# B&R Automation Studio project ACP180_Test
Automation Studio 4.12.5.95 SP; technology packages: mappMotion 5.26.1, mappView 5.24.1

## Configuration APC910

CPU 5PC900.TS17-00, AutomationRuntime M4.93, Build 4.1.2, Safety 0.0, Vc V4.72.6

### Task classes (Cpu.sw)
```
Cyclic#1 (cycle 800 us, tolerance 0 us):
  ShCamCtr <- Prog.ShCamCtr.prg
  StartMove <- Prog.StartMove.prg
  vis <- Prog.vis.prg
Cyclic#2:
  VRotary <- Prog.VRotary.prg
DataObjects: McAcpSys
NcDataObjects: Cam <- CAM.Cam.dob, McDriveLog
Binaries: arsvcreg, udbdef, mvLoader, arflatprv, McProfGen, McAcpDrv, arcoal, FWRules, TCData, McAcpSim, Config_1, ashwac, User, Config_4, sysconf, asfw, arconfig, iomap, Config_3, ashwd, Config_2, Role
Libraries: McBase, MpBase, McAxis, McAcpTrak, MpAxis, McAcpAx, AsBrStr, McPureVAx, arssl, astime, asieccon, powerlnk, runtime, fileio, asepl, sys_lib
```

### Hardware
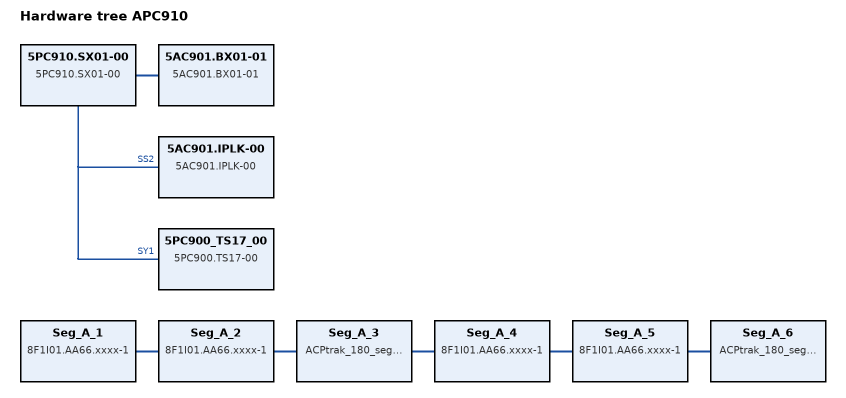
```
5AC901.BX01-01 : 5AC901.BX01-01 v1.1.0.0  [SY -> 5PC910.SX01-00.SY3]
5AC901.IPLK-00 : 5AC901.IPLK-00 v1.8.0.1  [SS -> 5PC910.SX01-00.SS2]
  Connector IF1:
    CycleTime = 800
    EplNatSubnet = 192.168.102.0
5PC900_TS17_00 : 5PC900.TS17-00 v2.1.0.0  [SY -> 5PC910.SX01-00.SY1]
  ConfigurationID = ACP180_Test_APC910
  Simulation = 1
  MotionLoggerSize = 2048000
  SystemTick = 800
  TaskClassIdleTime = 800
  Cyclic1Duration = 800
  Cyclic1Tolerance = 0
  Cyclic3Duration = 49600
  Cyclic3Tolerance = 49600
  Cyclic8Duration = 9600
  FileDevice1
  FileDeviceName1 = SvgData
  FileDevicePath1 = D:\Trak
  ActivateOpcUa = 1
  OpcUaInformationModels_PV_Version = 1
5PC910.SX01-00 : 5PC910.SX01-00 v2.1.0.0
  Connector IF1:
    AssignedOperatingSystem = ARemb
  Connector IF3:
    AssignedOperatingSystem = ARemb
    ActivateDevice = 1
  Connector IF4:
    AssignedOperatingSystem = ARemb
    ActivateDevice = 1
  Connector IF5:
    AssignedOperatingSystem = ARemb
  Connector IF6:
    AssignedOperatingSystem = ARemb
  Connector IF7:
    AssignedOperatingSystem = ARemb
  Connector IF8:
    AssignedOperatingSystem = ARemb
  Connector IF9:
    AssignedOperatingSystem = ARemb
Seg_A_1 : 8F1I01.AA66.xxxx-1 v1.0.0.2  [PLK2 -> Seg_A_2.PLK1 (NodeNumber=1) [Cable Type=PowerlinkCable, Length=10, Version=1.0.0.3]; PLK3 -> 5AC901.IPLK-00.IF1 (NodeNumber=1) [Cable Type=PowerlinkCable, Length=10, Version=1.0.0.3]]
  DriveConfiguration:
    McTypeID = LLMConfig
  DriveConfiguration/Segment:
    Shape = STRAIGHT660
    SegmentReference = Seg_A_1
    SegmentSectorDirection = Positive
    ElongationCompensation = UseAssemblySetting
    ACC = Inactive
    StopReaction = UseAssemblySetting
    SpeedFilter = UseAssemblySetting
    PositionControllerLagMonitor = UseAssemblySetting
Seg_A_2 : 8F1I01.AA66.xxxx-1 v1.0.0.2  [PLK1 -> Seg_A_1.PLK2 (NodeNumber=2) [Cable Type=PowerlinkCable, Length=10, Version=1.0.0.3]; PLK2 -> Seg_A_3.PLK1 (NodeNumber=2) [Cable Type=PowerlinkCable, Length=10, Version=1.0.0.3]]
  DriveConfiguration:
    McTypeID = LLMConfig
  DriveConfiguration/Segment:
    Shape = STRAIGHT660
    SegmentReference = Seg_A_2
    SegmentSectorDirection = Positive
    ElongationCompensation = UseAssemblySetting
    ACC = Inactive
    StopReaction = UseAssemblySetting
    SpeedFilter = UseAssemblySetting
    PositionControllerLagMonitor = UseAssemblySetting
Seg_A_3 : ACPtrak_180_seg_compact v0.0.0.6  [PLK1 -> Seg_A_2.PLK2 (NodeNumber=3) [Cable Type=PowerlinkCable, Length=10, Version=1.0.0.3]; PLK2 -> Seg_A_4.PLK1 (NodeNumber=3) [Cable Type=PowerlinkCable, Length=10, Version=1.0.0.3]]
  DriveConfiguration:
    McTypeID = LLMConfig
  DriveConfiguration/Segment:
    Shape = COMPACT_CURVE180
    SegmentReference = Seg_A_3
    SegmentSectorDirection = Positive
    ElongationCompensation = UseAssemblySetting
    ACC = Inactive
    StopReaction = UseAssemblySetting
    SpeedFilter = UseAssemblySetting
    PositionControllerLagMonitor = UseAssemblySetting
Seg_A_4 : 8F1I01.AA66.xxxx-1 v1.0.0.2  [PLK1 -> Seg_A_3.PLK2 (NodeNumber=4) [Cable Type=PowerlinkCable, Length=10, Version=1.0.0.3]; PLK2 -> Seg_A_5.PLK1 (NodeNumber=4) [Cable Type=PowerlinkCable, Length=10, Version=1.0.0.3]]
  DriveConfiguration:
    McTypeID = LLMConfig
  DriveConfiguration/Segment:
    Shape = STRAIGHT660
    SegmentReference = Seg_A_4
    SegmentSectorDirection = Positive
    ElongationCompensation = UseAssemblySetting
    ACC = Inactive
    StopReaction = UseAssemblySetting
    SpeedFilter = UseAssemblySetting
    PositionControllerLagMonitor = UseAssemblySetting
Seg_A_5 : 8F1I01.AA66.xxxx-1 v1.0.0.2  [PLK1 -> Seg_A_4.PLK2 (NodeNumber=5) [Cable Type=PowerlinkCable, Length=10, Version=1.0.0.3]; PLK2 -> Seg_A_6.PLK1 (NodeNumber=5) [Cable Type=PowerlinkCable, Length=10, Version=1.0.0.3]]
  DriveConfiguration:
    McTypeID = LLMConfig
  DriveConfiguration/Segment:
    Shape = STRAIGHT660
    SegmentReference = Seg_A_5
    SegmentSectorDirection = Positive
    ElongationCompensation = UseAssemblySetting
    ACC = Inactive
    StopReaction = UseAssemblySetting
    SpeedFilter = UseAssemblySetting
    PositionControllerLagMonitor = UseAssemblySetting
Seg_A_6 : ACPtrak_180_seg_compact v0.0.0.6  [PLK1 -> Seg_A_5.PLK2 (NodeNumber=6) [Cable Type=PowerlinkCable, Length=10, Version=1.0.0.3]]
  DriveConfiguration:
    McTypeID = LLMConfig
  DriveConfiguration/Segment:
    Shape = COMPACT_CURVE180
    SegmentReference = Seg_A_6
    SegmentSectorDirection = Positive
    ElongationCompensation = UseAssemblySetting
    ACC = Inactive
    StopReaction = UseAssemblySetting
    SpeedFilter = UseAssemblySetting
    PositionControllerLagMonitor = UseAssemblySetting
```

### Config_8.camlist - 5PC900_TS17_00/mappMotion/Config_8.camlist
```
Element CamList_1 (Type=camlist)
  Row[1]:
    CamName = Cam
    CamID = 1
    Description
```

### Config_7.axis - 5PC900_TS17_00/mappMotion/PureVAxis/Config_7.axis
```
Element gAxis_1 (Type=axis)
  BaseTypeIsReadOnly = 0
  BaseType = LinearBounded
    MeasurementUnit = 5066068
    MeasurementResolutionIsReadOnly = 0
    MeasurementResolution = 0.01
    CountDirectionIsReadOnly = 0
    CountDirection = Standard
  MovementLimitsIsReadOnly = 0
  MovementLimits = Internal
    Position:
      LowerLimitMin = -1.79769313486231E308
      UpperLimitMax = 1.79769313486231E308
      LowerLimit = -1000.0
      UpperLimit = 1000.0
    VelocityIsReadOnly = 0
    Velocity:
      VelocityMax = 3.4E38
      Velocity = 10.0
    AccelerationIsReadOnly = 0
    Acceleration:
      AccelerationMax = 3.4E38
      Acceleration = 50.0
    DecelerationIsReadOnly = 0
    Deceleration:
      DecelerationMax = 3.4E38
      Deceleration = 50.0
  Alarms = None
```

### Config_9.purevaxcfg - 5PC900_TS17_00/mappMotion/PureVAxis/Config_9.purevaxcfg
```
Element PureVAxCfg_1 (Type=purevaxcfg)
  TypeID = PureVAxConfig
  PureVAxis:
    AxisReference = gAxis_1
```

### Config_1.assembly - 5PC900_TS17_00/mappMotion/TrakOval/Config_1.assembly
```
Element gAssembly_1 (Type=assembly)
  Tracks:
    TrackSeparation = 0.030
    Track[1]:
      Segments:
        SegmentRef[1] = ::Seg_A_1
        SegmentRef[2] = ::Seg_A_2
        SegmentRef[3] = ::Seg_A_3
        SegmentRef[4] = ::Seg_A_4
        SegmentRef[5] = ::Seg_A_5
        SegmentRef[6] = ::Seg_A_6
      Position = Absolute
        SegmentRef = ::Seg_A_1
        SegmentCountDirection = RightToLeft
        Translation:
          X = 0.0
          Y = 0.0
          Z = 0.0
        Orientation:
          Angle1 = 0.0
          Angle2 = 0.0
          Angle3 = 180
  CommonSegmentSettings:
    SegmentSimulationOnPLC = Off
    CoggingCompensation = Active
      UpperVelLimit = 0.5
    ElongationCompensation = Inactive
    StopReaction = InductionHalt
    SpeedFilter = NotUsed
    ControllerParameters:
      DefaultParameter:
        Controller:
          Position:
            ProportionalGain = 200
          Speed:
            ProportionalGain = 80
            IntegrationTime = 0.0
          FeedForward:
            TotalMass = 1
            ForcePositive = 0.0
            ForceNegative = 0.0
            SpeedForceFactor = 0.0
            ForceLoad = 0.0
        MovementErrorLimits:
          PositionError = 0.001
          VelocityError = 0.05
        Diverter:
          ForceOverride = 1.0
      AdditionalParameterSets = NotUsed
    ScopeOfErrorReaction = Assembly
    ShuttleIdentificationTime = 0
    PositionControllerLagMonitor = Inactive
    Diverter:
      DiverterWeakEndOverrideFactor = 1.0
      DiverterStrenEndOverrideFactor = 1.0
  Shuttles:
    MaxShuttleCount = 25
    MaxShuttleCommandCount = 0
    Deceleration = 0.0
    UseConvoys = Inactive
    SwitchSectorAfterStop = SwitchOntoSegmentSector
      Scope = ShSs
    DistanceReserve:
      Collision = 0.002
      ErrorStop = 0.006
    ShuttleStereotypes:
      ShuttleStRef[1] = ShuttleStereotype_1
    MagnetPlateConfigurations:
      ShuttleType[1] = 8F1SA.100.xxxxxx-x
    CollisionAvoidance:
      Strategy = Constant
      Exclusion = NotUsed
      MaximumModelDimensions:
        Length:
          ExtentToFront = 0.025
          ExtentToBack = 0.025
        Width:
          Width = 0.040
    Coupling:
      CouplingFeature:
        EliminateShuttleToShuttleDelay = FALSE
  AssemblyFeatures:
    AssemblyFeatureRef[1] = AssemblyFeature_1
  Visualization:
    MonitoringPv = gShuttleMon
    ProcessingTaskClass = 1
  Alarms = None
```

### Config_10.axisfeature - 5PC900_TS17_00/mappMotion/TrakOval/Config_10.axisfeature
```
Element Feature_CamAutomat (Type=axisfeature)
  Type = CamAutomat
    CamAutomatType = ProfGen
      CommonParameters:
        Master:
          MasterSource = MasterAxis
            AxisReference
            ValueSource = SetPosition
            MaxVelocity = 1.0
          StartPosition = 0.0
          StartInterval = MasterAxisPeriod
        AdvancedParameters:
          StartStateParameters:
            StartState = 0
            RelMasterStartPos = 0.0
          AdditiveAxes:
            AdditiveMasterSource = NotUsed
            AdditiveSlaveSource = NotUsed
          MasterStartPositionMode = NotEvaluatedAnew
          ControlSettings:
            CrossLeftBoundary = PositionLimitedHorizontal
            CamChangeImmediately = CurrentMasterMoveDir
          StartIntervals
      States:
        State0 = Used
```

### Config_3.sector - 5PC900_TS17_00/mappMotion/TrakOval/Config_3.sector
```
Element SectorTrackA (Type=sector)
  Type = Composed
    StartSegment:
      SegmentRef = ::Seg_A_1
    IntermediateSegments:
      SegmentRef[1] = ::Seg_A_2
      SegmentRef[2] = ::Seg_A_3
      SegmentRef[3] = ::Seg_A_4
      SegmentRef[4] = ::Seg_A_5
    EndSegment:
      SegmentRef = ::Seg_A_6
      PositionRelativeTo = FromEnd
  Alarms = None
```

### Config_4.assemblyfeature - 5PC900_TS17_00/mappMotion/TrakOval/Config_4.assemblyfeature
```
Element AssemblyFeature_1 (Type=assemblyfeature)
  Type = InitShuttleSim
    InitShuttleSim[1]:
      SectorRef = SectorTrackA
      Orientation = Positive
      ShuttleDefinition = SingleShuttleDefinition
        Position[1] = 0.15
        Position[2] = 0.3
        Position[3] = 0.45
        Position[4] = 0.6
        Position[5] = 0.75
        Position[6] = 0.9
        Position[7] = 1.05
        Position[8] = 1.2
        Position[9] = 1.35
        Position[10] = 1.5
```

### Config_5.assemblyfeature - 5PC900_TS17_00/mappMotion/TrakOval/Config_5.assemblyfeature
```
Element AssemblyFeature_2 (Type=assemblyfeature)
  Type = Coupling
    CouplingObject[1]:
      Name = myCoupling
      ShuttleCount = 10
      CamAutomat
      CamList
```

### Config_6.processpointlist - 5PC900_TS17_00/mappMotion/TrakOval/Config_6.processpointlist
```
Element ProcessPointList_1 (Type=processpointlist)
  ProcessPoint[0]:
    Name = CamStartPoint
    SectorRef = SectorTrackA
    TriggerEventBufferSize = 10
    BarrierFunctionality = Off
  ProcessPoint[1]:
    Name = CamStopPoint
    SectorRef = SectorTrackA
    TriggerEventBufferSize = 10
    BarrierFunctionality = Off
```

## Logical view

Binary libraries used (declarations not repeated): operator, runtime, astime, AsIecCon, McBase, MpBase, McAxis, McAcpTrak, MpAxis, McAcpAx, AsBrStr, McPureVAx 5.26.1

### Global.typ - Global data types
```iecst
(* Shuttle user data structure *)

TYPE
	ShuttleUserData_type : 	STRUCT
		Color : ShuttleColor_enum; (* Example: product colour *)
		Weight : REAL; (* Example: product weight *)
		PartNumber : UDINT; (* Example: product part number *)
	END_STRUCT;
	ShuttleColor_enum :
		(
		ORANGE,
		GREEN,
		RED,
		BLUE,
		WHITE
		);
END_TYPE

(* Assembly interface *)

TYPE
	TrakAsmCommand_type : 	STRUCT
		Power : BOOL;
		ShuttleStart : BOOL;
		ShuttleStop : BOOL;
		Reset : BOOL;
	END_STRUCT;
	TrakAsmParameter_type : 	STRUCT
		Velocity : REAL;
		Acceleration : REAL;
		Deceleration : REAL;
	END_STRUCT;
	TrakAsmStatus_type : 	STRUCT
		Disabled : BOOL;
		Ready : BOOL;
		Homing : BOOL;
		Stopping : BOOL;
		ErrorStop : BOOL;
	END_STRUCT;
	TrakAsm_type : 	STRUCT
		Command : TrakAsmCommand_type;
		Parameter : TrakAsmParameter_type;
		Status : TrakAsmStatus_type;
		ShuttleCnt : UINT;
	END_STRUCT;
END_TYPE

(*Rotary Interface*)

TYPE
	RotaryCommand_type : 	STRUCT
		Power : BOOL;
		Update : BOOL;
		Home : BOOL;
		ErrorReset : BOOL;
		MoveVelocity : BOOL;
	END_STRUCT;
	RotaryStatus_type : 	STRUCT
		PowerOn : BOOL;
		Position : LREAL;
		Velocity : REAL;
		IsHomed : BOOL;
		InVelocity : BOOL;
		InPosition : BOOL;
		MoveActive : BOOL;
		Info : MpAxisBasicInfoType;
	END_STRUCT;
	RotaryPar_type : 	STRUCT
		Acceleration : REAL;
		Deceleration : REAL;
		Velocity : REAL;
	END_STRUCT;
	Rotary_type : 	STRUCT
		cmd : RotaryCommand_type;
		sts : RotaryStatus_type;
		par : RotaryPar_type;
	END_STRUCT;
END_TYPE
```

### Global.var - Global variables
```iecst
(* Assembly interface *)
VAR
	gTrakAsm : TrakAsm_type;
END_VAR
(* Shuttle user data structure *)
VAR
	gShuttleUserData : ShuttleUserData_type;
END_VAR
(* Shuttle monitor structure for Vis *)
VAR
	gShuttleMon : McAcpTrakAssemblyMonData;
END_VAR
(*Rotary Interface*)
VAR
	gRotary : Rotary_type;
END_VAR
```


### Program Logical/Prog/StartMove (IEC)

#### Types.typ
```iecst
TYPE
	StepEnum :
		(
		POWER_OFF,
		WAIT_POWER_OFF,
		POWERED_OFF,
		POWER_ON,
		WAIT_POWER_ON,
		GET_SHUTTLE,
		READY,
		START_MOVEMENT,
		WAIT_START_MOVEMENT,
		MOVING,
		STOPPING,
		WAIT_STOPPING,
		ERROR,
		RESET
	);
END_TYPE
```

#### Variables.var
```iecst
(* Constants *)
VAR CONSTANT
	MAX_SHUTTLE_CNT : USINT := 25; (* Maximum number of shuttles handled by the assembly *)
END_VAR
(* Sequence control *)
VAR
	Step : StepEnum;
	CurrentShuttleNumber : UINT;
	ShuttleReferences : ARRAY[1..MAX_SHUTTLE_CNT] OF McAxisType;
	UserDataSize : UDINT;
END_VAR
(* Function blocks *)
VAR
	MC_BR_AsmPowerOn_AcpTrak_0 : MC_BR_AsmPowerOn_AcpTrak;
	MC_BR_AsmPowerOff_AcpTrak_0 : MC_BR_AsmPowerOff_AcpTrak;
	MC_BR_AsmGetShuttle_AcpTrak_0 : MC_BR_AsmGetShuttle_AcpTrak;
	MC_BR_AsmStop_AcpTrak_0 : MC_BR_AsmStop_AcpTrak;
	MC_BR_AsmReadStatus_AcpTrak_0 : MC_BR_AsmReadStatus_AcpTrak;
	MC_BR_AsmReset_AcpTrak_0 : MC_BR_AsmReset_AcpTrak;
	MC_BR_RoutedMoveVel_AcpTrak_0 : MC_BR_RoutedMoveVel_AcpTrak;
END_VAR
(*CAM Control*)
```

#### Main.st
```iecst
PROGRAM _INIT
    (* Initialize parameters for shuttle movements. *)
	gTrakAsm.Parameter.Velocity := 1.0;
	gTrakAsm.Parameter.Acceleration := 10.0;
	gTrakAsm.Parameter.Deceleration := 10.0;

	(* Write this value into the size of user data in the shuttle stereotype configuration. *)
	UserDataSize := SIZEOF(gShuttleUserData);

	(* Set the assembly reference for all assembly function blocks. *)
	MC_BR_AsmPowerOn_AcpTrak_0.Assembly     := ADR(gAssembly_1);
	MC_BR_AsmPowerOff_AcpTrak_0.Assembly    := ADR(gAssembly_1);
	MC_BR_AsmStop_AcpTrak_0.Assembly        := ADR(gAssembly_1);
	MC_BR_AsmGetShuttle_AcpTrak_0.Assembly  := ADR(gAssembly_1);
	MC_BR_AsmReadStatus_AcpTrak_0.Assembly  := ADR(gAssembly_1);
	MC_BR_AsmReset_AcpTrak_0.Assembly       := ADR(gAssembly_1);

	(* Enable reading of current status of the assembly. *)
	MC_BR_AsmReadStatus_AcpTrak_0.Enable := TRUE;

	(* Initialize constant parameters for routed moves. *)
	MC_BR_RoutedMoveVel_AcpTrak_0.Sector        := ADR(SectorTrackA);
	MC_BR_RoutedMoveVel_AcpTrak_0.Jerk          := 0.0;
	MC_BR_RoutedMoveVel_AcpTrak_0.BufferMode    := mcABORTING;
	MC_BR_RoutedMoveVel_AcpTrak_0.AdvancedParameters.StartDirection     := mcDIR_UNDEFINED;
	MC_BR_RoutedMoveVel_AcpTrak_0.AdvancedParameters.EndDirection       := mcDIR_POSITIVE;
	MC_BR_RoutedMoveVel_AcpTrak_0.AdvancedParameters.ShuttleOrientation := mcDIR_UNDEFINED;

	(* Initialize constant parameter for assembly stop command. *)
//	MC_BR_AsmStop_AcpTrak_0.AdvancedParameters.StopMode := mcSTOPMODE_JERK_LIMIT;
END_PROGRAM

PROGRAM _CYCLIC

	gRotary;

	IF gTrakAsm.Status.ErrorStop THEN
		Step := ERROR;
	END_IF

	CASE Step OF

		(* Power off assembly and wait for power on command *)
		POWER_OFF:
			(* Assembly is already powered off. *)
			IF gTrakAsm.Status.Disabled THEN
				Step := POWERED_OFF;
			ELSE
				MC_BR_AsmPowerOff_AcpTrak_0.Execute := TRUE;
				Step := WAIT_POWER_OFF;
			END_IF

			(* The assembly is being powered off. *)
		WAIT_POWER_OFF:
			(* Power off is done. *)
			IF MC_BR_AsmPowerOff_AcpTrak_0.Done THEN
				MC_BR_AsmPowerOff_AcpTrak_0.Execute := FALSE;
				Step := POWERED_OFF;
			ELSIF MC_BR_AsmPowerOff_AcpTrak_0.Error THEN
				Step := ERROR;
			END_IF

			(* The assembly is powered off, wait for a command to power it on. *)
		POWERED_OFF:
			(* The assembly is to be powered on. *)
			IF gTrakAsm.Command.Power THEN
				Step := POWER_ON;
			END_IF

			(* Power on assembly *)
		POWER_ON:
			MC_BR_AsmPowerOn_AcpTrak_0.Execute := TRUE;
			Step := WAIT_POWER_ON;

			(* The assembly is being powered on. *)
		WAIT_POWER_ON:
			(* Assembly is not yet powered on. *)
			IF MC_BR_AsmPowerOn_AcpTrak_0.Done THEN
				MC_BR_AsmPowerOn_AcpTrak_0.Execute := FALSE;

				(* Store the shuttles in the shuttle array. On real hardware, the set of shuttles might have changed. *)
				CurrentShuttleNumber := 1;
				brsmemset(ADR(ShuttleReferences), 0, SIZEOF(ShuttleReferences));
				Step := GET_SHUTTLE;
			ELSIF MC_BR_AsmPowerOn_AcpTrak_0.Error THEN
				Step := ERROR;
			END_IF

			(* Get all shuttles on the assembly (those physically available on the real hardware or the added ones in the simulation, resp.). *)
		GET_SHUTTLE:
			MC_BR_AsmGetShuttle_AcpTrak_0.Enable := TRUE;

			IF MC_BR_AsmGetShuttle_AcpTrak_0.Valid THEN
				(* There are no shuttles on the assembly. *)
				IF MC_BR_AsmGetShuttle_AcpTrak_0.TotalCount = 0 THEN
					gTrakAsm.ShuttleCnt := 0;
					MC_BR_AsmGetShuttle_AcpTrak_0.Enable := FALSE;
					MC_BR_AsmGetShuttle_AcpTrak_0.Next := FALSE;

					Step := READY;
                (* As soon as the next shuttle has been output by the function block, RemainingCount
                   is reduced and this condition becomes true. *)
				ELSIF (MC_BR_AsmGetShuttle_AcpTrak_0.RemainingCount <> (MC_BR_AsmGetShuttle_AcpTrak_0.TotalCount - CurrentShuttleNumber)) THEN
					CurrentShuttleNumber := CurrentShuttleNumber + 1;
					MC_BR_AsmGetShuttle_AcpTrak_0.Next := FALSE;
				ELSE
					(* Store all axis references in an array for global movement commands. *)
					ShuttleReferences[CurrentShuttleNumber] := MC_BR_AsmGetShuttle_AcpTrak_0.Axis;
					(* Get next shuttle reference with positive edge on .Next. *)
					MC_BR_AsmGetShuttle_AcpTrak_0.Next := TRUE;

					(* All shuttles have been stored. *)
					IF (MC_BR_AsmGetShuttle_AcpTrak_0.RemainingCount = 0) THEN
						gTrakAsm.ShuttleCnt := MC_BR_AsmGetShuttle_AcpTrak_0.TotalCount;
						MC_BR_AsmGetShuttle_AcpTrak_0.Enable := FALSE;
						MC_BR_AsmGetShuttle_AcpTrak_0.Next := FALSE;

						Step := READY;
					END_IF
				END_IF
			END_IF

			(* Assembly is active and ready for movement. *)
		READY:
			(* Power off the assembly. *)
			IF NOT gTrakAsm.Command.Power THEN
				Step := POWER_OFF;
				(* Wait for movement command if shuttles are present. *)
			ELSIF gTrakAsm.Command.ShuttleStart AND gTrakAsm.ShuttleCnt > 0 THEN
				gTrakAsm.Command.ShuttleStart := FALSE;
				CurrentShuttleNumber := 1;
				Step := START_MOVEMENT;
			END_IF

			(* Move all shuttles on assembly to the same target position with the same velocity. *)
			(* Used for startup to accelerate all shuttles to an initial velocity in order to
			pass the first process-point. *)
		START_MOVEMENT:
			IF CurrentShuttleNumber <= gTrakAsm.ShuttleCnt THEN
				MC_BR_RoutedMoveVel_AcpTrak_0.Axis          := ADR(ShuttleReferences[CurrentShuttleNumber]);
				MC_BR_RoutedMoveVel_AcpTrak_0.Position      := 0.3 + gTrakAsm.ShuttleCnt * 0.15;
				MC_BR_RoutedMoveVel_AcpTrak_0.Velocity      := gTrakAsm.Parameter.Velocity;
				MC_BR_RoutedMoveVel_AcpTrak_0.RouteVelocity := gTrakAsm.Parameter.Velocity;
				MC_BR_RoutedMoveVel_AcpTrak_0.Acceleration  := gTrakAsm.Parameter.Acceleration;
				MC_BR_RoutedMoveVel_AcpTrak_0.Deceleration  := gTrakAsm.Parameter.Deceleration;
				MC_BR_RoutedMoveVel_AcpTrak_0.Execute       := TRUE;

				Step := WAIT_START_MOVEMENT;
			ELSE
				Step := MOVING;
			END_IF

			(* Wait until a shuttle movement is active. *)
		WAIT_START_MOVEMENT:
			IF MC_BR_RoutedMoveVel_AcpTrak_0.Active THEN
				MC_BR_RoutedMoveVel_AcpTrak_0.Execute := FALSE;
				CurrentShuttleNumber := CurrentShuttleNumber + 1;
				Step := START_MOVEMENT;
				(* There is invalid speed or acceleration setting or shuttle caused an error stop. *)
			ELSIF MC_BR_RoutedMoveVel_AcpTrak_0.Error THEN
				Step := ERROR;
			END_IF

			(* A movement has been started for all shuttles. *)
		MOVING:
			(* Wait for Stop command. *)
			IF gTrakAsm.Command.ShuttleStop THEN
				gTrakAsm.Command.ShuttleStop := FALSE;
				Step := STOPPING;
			END_IF

			(* Stop all shuttles with specified deceleration at their current locations. *)
		STOPPING:
			MC_BR_AsmStop_AcpTrak_0.Execute := TRUE;
			Step := WAIT_STOPPING;

			(* Wait until all shuttles are stopped. *)
		WAIT_STOPPING:
			IF MC_BR_AsmStop_AcpTrak_0.Done THEN
				MC_BR_AsmStop_AcpTrak_0.Execute := FALSE;
				Step := READY;
				(* A shuttle caused an error stop. *)
			ELSIF MC_BR_AsmStop_AcpTrak_0.Error THEN
				Step := ERROR;
			END_IF

			(* An error occured on the assembly. *)
		ERROR:
			(* Wait for the user to trigger the error reset. *)
			IF gTrakAsm.Command.Reset THEN
				gTrakAsm.Command.Reset := FALSE;
				MC_BR_AsmReset_AcpTrak_0.Execute := TRUE;
				Step := RESET;
			END_IF

			(* Reset assembly due to an error. *)
		RESET:
			IF MC_BR_AsmReset_AcpTrak_0.Done THEN
				gTrakAsm.Command.ShuttleStart           := FALSE;
				gTrakAsm.Command.ShuttleStop            := FALSE;
				MC_BR_AsmReset_AcpTrak_0.Execute        := FALSE;
				MC_BR_AsmPowerOn_AcpTrak_0.Execute      := FALSE;
				MC_BR_AsmPowerOff_AcpTrak_0.Execute     := FALSE;
				MC_BR_AsmStop_AcpTrak_0.Execute         := FALSE;
				MC_BR_RoutedMoveVel_AcpTrak_0.Execute   := FALSE;

				Step := READY;
			END_IF
	END_CASE

	(* Read assembly status cyclically to assembly interface. *)
	gTrakAsm.Status.Disabled  := MC_BR_AsmReadStatus_AcpTrak_0.AssemblyDisabled;
	gTrakAsm.Status.Ready     := MC_BR_AsmReadStatus_AcpTrak_0.AssemblyReady;
	gTrakAsm.Status.Homing    := MC_BR_AsmReadStatus_AcpTrak_0.AssemblyHoming;
	gTrakAsm.Status.Stopping  := MC_BR_AsmReadStatus_AcpTrak_0.AssemblyStopping;
	gTrakAsm.Status.ErrorStop := MC_BR_AsmReadStatus_AcpTrak_0.AssemblyErrorStop;

	(* Cyclic function blocks calls *)
	MC_BR_AsmPowerOn_AcpTrak_0();
	MC_BR_AsmGetShuttle_AcpTrak_0();
	MC_BR_AsmPowerOff_AcpTrak_0();
	MC_BR_AsmStop_AcpTrak_0();
	MC_BR_RoutedMoveVel_AcpTrak_0();
	MC_BR_AsmReadStatus_AcpTrak_0();
	MC_BR_AsmReset_AcpTrak_0();
END_PROGRAM
```

### Program Logical/Prog/vis (IEC)

#### Variables.var
```iecst
VAR
	Vis : McAcpTrakAssemblyVisData;
	SizeOfVis : UDINT := 0;
	VisShuttleCnt : USINT := 0;
	i : USINT := 0;
	UserData : REFERENCE TO ShuttleUserData_type;
END_VAR
```

#### Main.st
```iecst
PROGRAM _INIT
    (* Size of Vis structure - this value has to be entered in B&R scene viewer (PVI -> Options -> Size) *)
	SizeOfVis := SIZEOF(Vis);
	(* Maximum number of displayed shuttles *)
	VisShuttleCnt := SIZEOF(Vis.Shuttle) / SIZEOF(Vis.Shuttle[0]);
END_PROGRAM

PROGRAM _CYCLIC
	FOR i := 0 TO (VisShuttleCnt - 1) DO
		IF gShuttleMon.Shuttle[i].Available THEN
			(* Format selected monitor data to fit B&R scene viewer. *)
			Vis.Shuttle[i].Available     := 1;
			Vis.Shuttle[i].PositionX     := LREAL_TO_REAL(gShuttleMon.Shuttle[i].Position.X);
			Vis.Shuttle[i].PositionY     := LREAL_TO_REAL(gShuttleMon.Shuttle[i].Position.Y);
			Vis.Shuttle[i].RotationZ     := LREAL_TO_REAL(gShuttleMon.Shuttle[i].Orientation.Angle1);
			Vis.Shuttle[i].ExtentToFront := LREAL_TO_REAL(gShuttleMon.Shuttle[i].ExtentToFront);
			Vis.Shuttle[i].ExtentToBack  := LREAL_TO_REAL(gShuttleMon.Shuttle[i].ExtentToBack);
			Vis.Shuttle[i].Width         := LREAL_TO_REAL(gShuttleMon.Shuttle[i].Width);
			brsitoa(gShuttleMon.Shuttle[i].Index, ADR(Vis.Shuttle[i].Text));

			(* Color is defined with RGB values between 0 and 1. The default shuttle color is gray. *)
			Vis.Shuttle[i].ColorRed      := 0.5;
			Vis.Shuttle[i].ColorGreen    := 0.5;
			Vis.Shuttle[i].ColorBlue     := 0.5;

			(* Example: Set shuttle colour via user data. *)
			IF gShuttleMon.Shuttle[i].UserData <> 0 THEN
				(* Set access to user data of this shuttle. *)
				UserData ACCESS gShuttleMon.Shuttle[i].UserData;

				(* Set RGB values for specific colors. *)
				IF UserData.Color = ORANGE THEN
					Vis.Shuttle[i].ColorRed     := 1.000;
					Vis.Shuttle[i].ColorGreen   := 0.5451;
					Vis.Shuttle[i].ColorBlue    := 0.000;
				ELSIF UserData.Color = GREEN THEN
					Vis.Shuttle[i].ColorRed     := 0.000;
					Vis.Shuttle[i].ColorGreen   := 1.000;
					Vis.Shuttle[i].ColorBlue    := 0.000;
				ELSIF UserData.Color = RED THEN
					Vis.Shuttle[i].ColorRed     := 1.000;
					Vis.Shuttle[i].ColorGreen   := 0.000;
					Vis.Shuttle[i].ColorBlue    := 0.000;
				ELSIF UserData.Color = BLUE THEN
					Vis.Shuttle[i].ColorRed     := 0.000;
					Vis.Shuttle[i].ColorGreen   := 0.000;
					Vis.Shuttle[i].ColorBlue    := 1.000;
				ELSIF UserData.Color = WHITE THEN
					Vis.Shuttle[i].ColorRed     := 1.000;
					Vis.Shuttle[i].ColorGreen   := 1.000;
					Vis.Shuttle[i].ColorBlue    := 1.000;
				END_IF
			END_IF
		ELSE
			(* If the selected shuttle is not available, it will be invisible in the Scene Viewer. *)
			brsmemset(ADR(Vis.Shuttle[i]), 0, SIZEOF(Vis.Shuttle[0]));
		END_IF
	END_FOR
END_PROGRAM
```

### Program Logical/Prog/ShCamCtr (IEC)

#### Main.st
```iecst
PROGRAM _INIT
	(* Insert code here *)

END_PROGRAM

PROGRAM _CYCLIC
	(* Insert code here *)

END_PROGRAM

PROGRAM _EXIT
	(* Insert code here *)

END_PROGRAM
```

### Program Logical/Prog/VRotary (IEC)

#### Variables.var
```iecst
VAR
	fbMpAxisBasic : MpAxisBasic;
	MpAxisBasicPar : MpAxisBasicParType;
END_VAR
```

#### Main.st
```iecst
PROGRAM _INIT
	(* Insert code here *)

	gRotary.par.Acceleration := 10;
	gRotary.par.Deceleration := 10;
	gRotary.par.Velocity := 1.5;

	MpAxisBasicPar.Acceleration := gRotary.par.Acceleration;
	MpAxisBasicPar.Deceleration := gRotary.par.Deceleration;
	MpAxisBasicPar.Velocity := gRotary.par.Velocity;

	fbMpAxisBasic.MpLink := ADR(gAxis_1);
	fbMpAxisBasic.Parameters := ADR(MpAxisBasicPar);
	fbMpAxisBasic.Enable := TRUE;
	fbMpAxisBasic();

END_PROGRAM

PROGRAM _CYCLIC
	(* Insert code here *)

	MpAxisBasicPar.Acceleration := gRotary.par.Acceleration;
	MpAxisBasicPar.Deceleration := gRotary.par.Deceleration;
	MpAxisBasicPar.Velocity := gRotary.par.Velocity;

	fbMpAxisBasic.Power := gRotary.cmd.Power;
	fbMpAxisBasic.Update := gRotary.cmd.Update;
	fbMpAxisBasic.Home := gRotary.cmd.Home;
	fbMpAxisBasic.MoveVelocity := gRotary.cmd.MoveVelocity;
	fbMpAxisBasic.ErrorReset := gRotary.cmd.ErrorReset;

	gRotary.sts.InPosition := fbMpAxisBasic.InPosition;
	gRotary.sts.PowerOn := fbMpAxisBasic.PowerOn;
	gRotary.sts.Position := fbMpAxisBasic.Position;
	gRotary.sts.Velocity := fbMpAxisBasic.Velocity;
	gRotary.sts.IsHomed := fbMpAxisBasic.IsHomed;
	gRotary.sts.InVelocity := fbMpAxisBasic.InVelocity;
	gRotary.sts.MoveActive := fbMpAxisBasic.MoveActive;
	gRotary.sts.Info := fbMpAxisBasic.Info;

	fbMpAxisBasic();
END_PROGRAM

PROGRAM _EXIT
	(* Insert code here *)
	 fbMpAxisBasic(Enable := FALSE);
END_PROGRAM
```

### Data object Logical/CAM/Cam (Cam)

#### Cam.cam - Cam for mapp Motion
```
CamProfile (NcManager=ACP10, MasterAxisVelocity=1, MasterAxisAcceleration=0, DefaultCurveType=Polynomial5, MathematicalNotation=true)
  Cam NewMotionObject1 (LeftBoundaryIndex=0, RightBoundaryIndex=0)
    Supremum (y=1.7e+308, Dy=1.7e+308, IsMathDy=true, Ddy=1.7e+308, IsMathDdy=true, Dddy=1.7e+308, IsMathDddy=true)
    Infimum (y=-1.7e+308, Dy=-1.7e+308, IsMathDy=true, Ddy=-1.7e+308, IsMathDdy=true, Dddy=1.7e+308, IsMathDddy=true)
```
